FUNCTION_BLOCK DummyControl (* Basic Function Block Type *)
  (* Standard: 61499-2 *)
  (* Version 0.0, 6/17/2016, Andrei, nxtControl GmbH, Template *)
  PACKAGE Main;
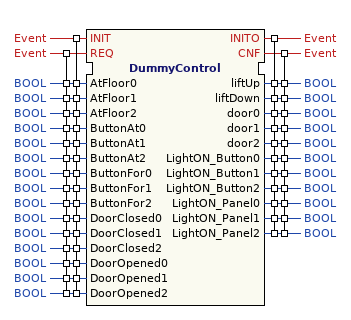
  EVENT_INPUT
    INIT WITH AtFloor0, AtFloor1, AtFloor2, DoorClosed0, DoorClosed1, DoorClosed2, ButtonAt0, ButtonAt1, ButtonAt2, ButtonFor0, ButtonFor1, ButtonFor2, DoorOpened0, DoorOpened1, DoorOpened2; (* Initialization Request *)
    REQ WITH AtFloor0, AtFloor1, AtFloor2, DoorClosed0, DoorClosed1, DoorClosed2, ButtonAt0, ButtonAt1, ButtonAt2, ButtonFor0, ButtonFor1, ButtonFor2, DoorOpened0, DoorOpened1, DoorOpened2; (* Normal Execution Request *)
  END_EVENT
  EVENT_OUTPUT
    INITO WITH liftUp, liftDown, door0, door1, door2, LightON_Button0, LightON_Button1, LightON_Button2, LightON_Panel0, LightON_Panel1, LightON_Panel2; (* Initialization Confirm *)
    CNF WITH liftUp, liftDown, door0, door1, door2, LightON_Button0, LightON_Button1, LightON_Button2, LightON_Panel0, LightON_Panel1, LightON_Panel2; (* Execution Confirmation *)
  END_EVENT
  VAR_INPUT
    AtFloor0 : BOOL; (* Input event qualifier *)
    AtFloor1 : BOOL;
    AtFloor2 : BOOL;
    ButtonAt0 : BOOL;
    ButtonAt1 : BOOL;
    ButtonAt2 : BOOL;
    ButtonFor0 : BOOL;
    ButtonFor1 : BOOL;
    ButtonFor2 : BOOL;
    DoorClosed0 : BOOL;
    DoorClosed1 : BOOL;
    DoorClosed2 : BOOL;
    DoorOpened0 : BOOL;
    DoorOpened1 : BOOL;
    DoorOpened2 : BOOL;
  END_VAR
  VAR_OUTPUT
    liftUp : BOOL;
    liftDown : BOOL; (* Output event qualifier *)
    door0 : BOOL;
    door1 : BOOL;
    door2 : BOOL;
    LightON_Button0 : BOOL;
    LightON_Button1 : BOOL;
    LightON_Button2 : BOOL;
    LightON_Panel0 : BOOL;
    LightON_Panel1 : BOOL;
    LightON_Panel2 : BOOL;
  END_VAR
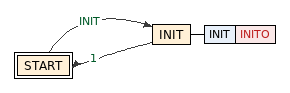
  EC_STATES
    START; (* Initial State *)
    INIT : INIT -> INITO;
  END_STATES
  EC_TRANSITIONS
    START TO INIT := INIT;
    INIT TO START := 1;
  END_TRANSITIONS
  ALGORITHM INIT IN ST: (* Initialization algorithm *)
;
  END_ALGORITHM
  ALGORITHM REQ IN ST: (* Normally executed algorithm *)
;
  END_ALGORITHM
END_FUNCTION_BLOCK
